{attribute 'qualified_only'}
{attribute 'strict'}
TYPE E_IndexedPositionTransitionRequest :
(
	NoRequest,
	ReceiveFromLeft,
	ReceiveFromRight,
	ReceiveFromFront,
	ReceiveFromRear,
	SendToLeft,
	SendToRight,
	SendToFront,
	SendToRear
);
END_TYPE

(* stored: Version 1.1.0.1, ProductVersion 3.1.4024.12
   DUT E_IndexedPositionTransitionRequest: Id {0ba08914-510c-4fc9-9197-e4d2090b6de2} *)
